(* PLC project Unnamed, Unknown Unnamed 1 *)
(* stored: creationDateTime 2024-07-13T14:13:31, modificationDateTime 2024-07-14T13:48:20 *)

PROGRAM program0
  VAR
    Y0 AT %IX100.0 : BOOL;
    Y1 AT %IX100.1 : BOOL;
    Y2 AT %IX100.2 : BOOL;
    Y3 AT %IX100.3 : BOOL;
    Y4 AT %IX100.4 : BOOL;
    D0 AT %QW104 : WORD;
    D1 AT %QW105 : WORD;
    D2 AT %QW106 : WORD;
    D3 AT %QW107 : WORD;
    M1 AT %IW100 : INT;
    M2 AT %IW101 : INT;
    M3 AT %IW102 : INT;
    M4 AT %IW103 : INT;
  END_VAR
  VAR
    TOF0 : TOF;
    TON0 : TON;
  END_VAR

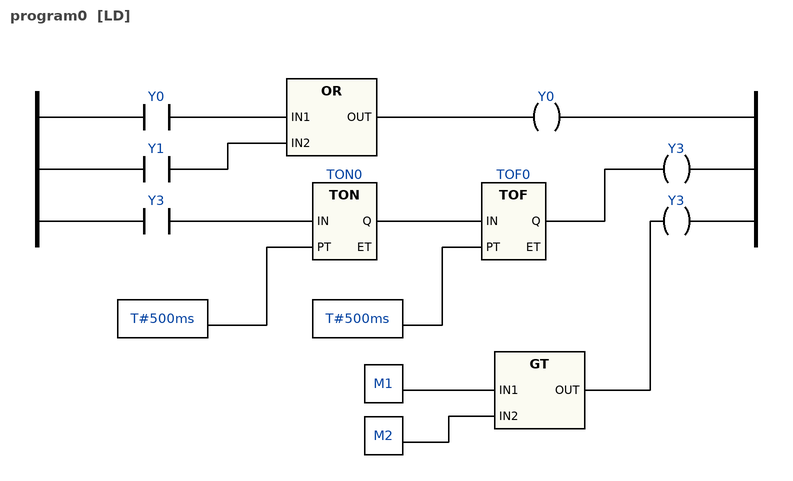
(* LD diagram, written out as Structured Text *)
Y0 := Y0 OR Y1;
TON0(IN := Y3, PT := T#500ms);
TOF0(IN := TON0.Q, PT := T#500ms);
Y3 := TOF0.Q;
Y3 := M1 > M2;
END_PROGRAM

CONFIGURATION Config0
  RESOURCE Res0 ON PLC
    TASK task0(INTERVAL := T#20ms, PRIORITY := 0);
    PROGRAM instance0 WITH task0 : program0;
  END_RESOURCE
END_CONFIGURATION
